{attribute 'qualified_only'}
{attribute 'strict'}
{attribute 'to_string'}
 
TYPE eConnectionState :
(
	disconnected := 0,			// no mqtt connection established
	connected	:= 1,			 // connected but not authorized yet
	authorization_declined := 2, // connected but authorization failed
	authorized	:= 3			// connected and authorized
);
END_TYPE

(* stored: Version 1.1.0.1, ProductVersion 3.1.4026.18
   DUT eConnectionState: Id {7f010d7f-b3e5-4466-9dc1-448e0a404b52} *)
